// Mitsubishi GX Works2 project: Main_plc_id_2   PLC: FX3U/FX3UC

PROGRAM MAIN
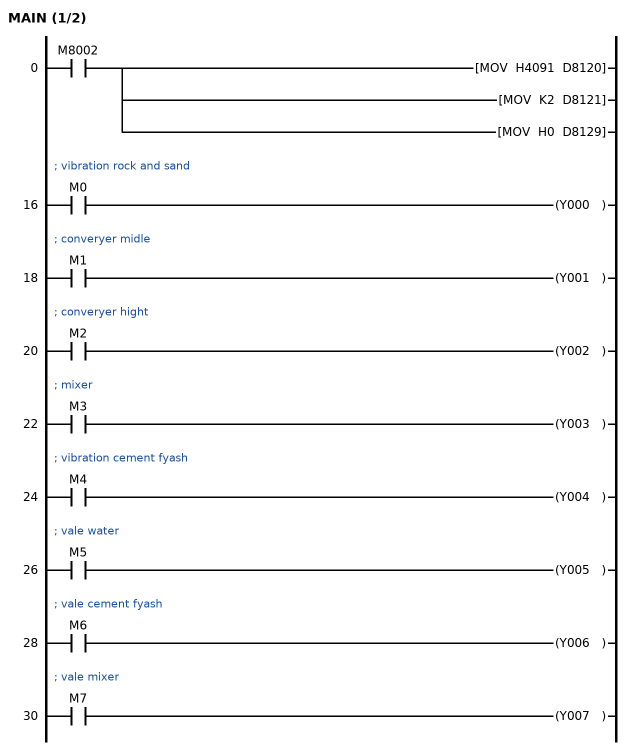
0     LD      M8002
      MOV     H4091 D8120
      MOV     K2 D8121
      MOV     H0 D8129
; vibration rock and sand
16    LD      M0
      OUT     Y000
; converyer midle
18    LD      M1
      OUT     Y001
; converyer hight
20    LD      M2
      OUT     Y002
; mixer
22    LD      M3
      OUT     Y003
; vibration cement fyash
24    LD      M4
      OUT     Y004
; vale water
26    LD      M5
      OUT     Y005
; vale cement fyash
28    LD      M6
      OUT     Y006
; vale mixer
30    LD      M7
      OUT     Y007
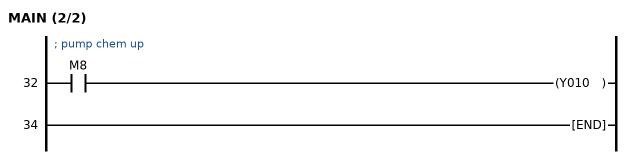
; pump chem up
32    LD      M8
      OUT     Y010
34    END
END_PROGRAM
